Staubli VAL3: Init.pgx

program Init()
  local num l_ni
  local string l_sKey
begin
  //
  bUserRefresh=bListRefresh=true
  //
  bExit=false
  //
  call readFileList(sFolder,sFileList)
  //按照前缀sDeli选择相应的文件
  //call selectFile(sDeli,sFileList)
  //

  //call getList(PublicData:sPrd,sPrd)

  resize(sPrd,1,size(PublicData:sPrd))
  for l_ni=0 to size(PublicData:sPrd)-1
    sPrd[l_ni]=PublicData:sPrd[l_ni]
  endFor

  resize(sProductList,1,size(PublicData:sProductList))
  for l_ni=0 to size(PublicData:sProductList)-1
    sProductList[l_ni]=PublicData:sProductList[l_ni]
  endFor

end
